// TIA Portal V16 export
FUNCTION_BLOCK "FB_PumpControl_LAD"   // FB2, LAD
{ S7_Optimized_Access := 'TRUE' }
// stored: AutoNumber true
   VAR_INPUT
      FirstScan : Bool;
      AutoMode : Bool;
      StartButton : Bool;
      StopOK : Bool;
      SafetyOK : Bool;
      OverloadOK : Bool;
      SourceWaterOK : Bool;
      LowWet : Bool;
      HighWet : Bool;
      ResetButton : Bool;
      MotorFeedback : Bool;
      MinOffTime : Time := T#5s;
      FeedbackTime : Time := T#3s;
      MaxRunTime : Time := T#10m;
   END_VAR
   VAR_OUTPUT
      PumpCmd : Bool;
      Alarm : Bool;
      Enabled : Bool;
      RunningConfirmed : Bool;
      FaultBits : Word;
      State : USInt;
   END_VAR
   VAR
      RunState : Bool := FALSE;
      EnableState : Bool := FALSE;
      FaultMemory : Word := W#16#0000;
      StartPrev : Bool;
      ResetPrev : Bool;
      AutoPrev : Bool;
      AutoDemand : Bool;
      ManualDemand : Bool;
      OffTimer : TON_TIME;
      RunTimer : TON_TIME;
      StartFeedbackTimer : TON_TIME;
      StopFeedbackTimer : TON_TIME;
   END_VAR
   VAR_TEMP
      StartPulse : Bool;
      ResetPulse : Bool;
      ModeChanged : Bool;
      SensorInvalid : Bool;
      ConfigInvalid : Bool;
      HealthyInputs : Bool;
      Demand : Bool;
      BadMinOff : Bool;
      BadFeedback : Bool;
      BadMaxRun : Bool;
      Disarm : Bool;
      StartAccepted : Bool;
   END_VAR
BEGIN

REGION Network 1: 01 - Startup: reset RunState
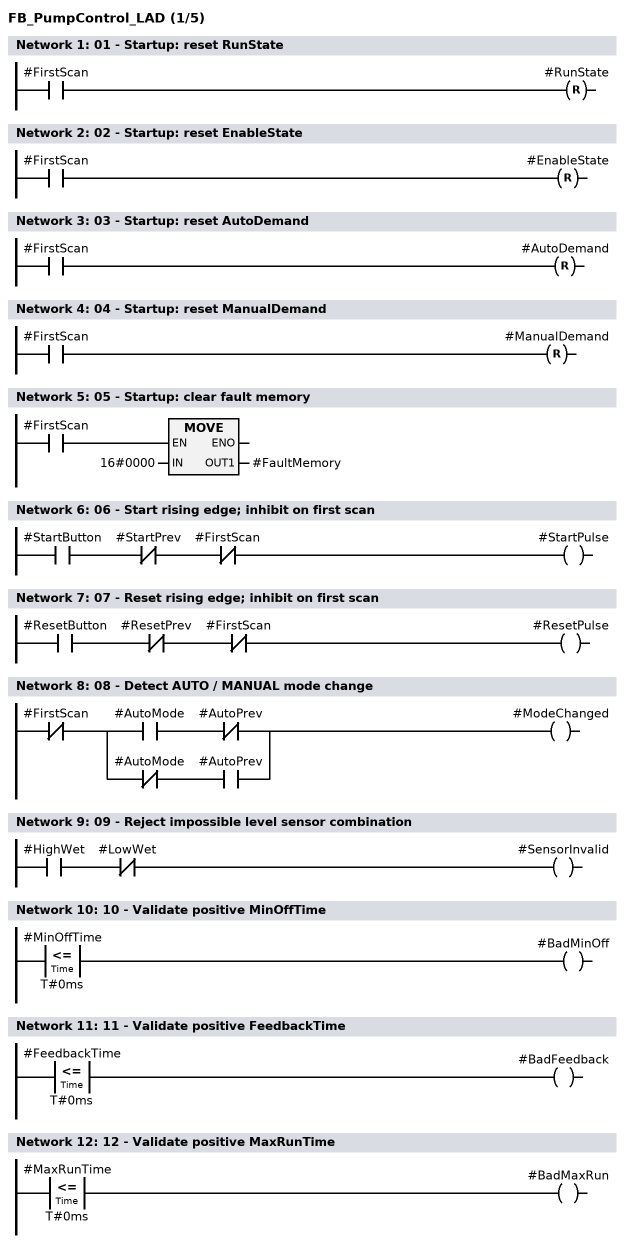
   RUNG wire#powerrail
      Contact( #FirstScan )
      R_Coil( #RunState )
   END_RUNG
   // the same network as SCL:
   IF #FirstScan THEN #RunState := FALSE; END_IF;
END_REGION

REGION Network 2: 02 - Startup: reset EnableState
   RUNG wire#powerrail
      Contact( #FirstScan )
      R_Coil( #EnableState )
   END_RUNG
   // the same network as SCL:
   IF #FirstScan THEN #EnableState := FALSE; END_IF;
END_REGION

REGION Network 3: 03 - Startup: reset AutoDemand
   RUNG wire#powerrail
      Contact( #FirstScan )
      R_Coil( #AutoDemand )
   END_RUNG
   // the same network as SCL:
   IF #FirstScan THEN #AutoDemand := FALSE; END_IF;
END_REGION

REGION Network 4: 04 - Startup: reset ManualDemand
   RUNG wire#powerrail
      Contact( #FirstScan )
      R_Coil( #ManualDemand )
   END_RUNG
   // the same network as SCL:
   IF #FirstScan THEN #ManualDemand := FALSE; END_IF;
END_REGION

REGION Network 5: 05 - Startup: clear fault memory
   RUNG wire#powerrail
      Contact( #FirstScan )
      { S7_GenerateENO := "TRUE" } Move(in := 16#0000, out1 => #FaultMemory)
   END_RUNG
   // the same network as SCL:
   IF #FirstScan THEN #FaultMemory := 16#0000; END_IF;
END_REGION

REGION Network 6: 06 - Start rising edge; inhibit on first scan
   RUNG wire#powerrail
      Contact( #StartButton )
      I_Contact( #StartPrev )
      I_Contact( #FirstScan )
      Coil( #StartPulse )
   END_RUNG
   // the same network as SCL:
   #StartPulse := #StartButton AND NOT #StartPrev AND NOT #FirstScan;
END_REGION

REGION Network 7: 07 - Reset rising edge; inhibit on first scan
   RUNG wire#powerrail
      Contact( #ResetButton )
      I_Contact( #ResetPrev )
      I_Contact( #FirstScan )
      Coil( #ResetPulse )
   END_RUNG
   // the same network as SCL:
   #ResetPulse := #ResetButton AND NOT #ResetPrev AND NOT #FirstScan;
END_REGION

REGION Network 8: 08 - Detect AUTO / MANUAL mode change
   RUNG wire#powerrail
      I_Contact( #FirstScan )
      wire#w1
      Contact( #AutoMode )
      I_Contact( #AutoPrev )
      wire#w2
      Coil( #ModeChanged )
   END_RUNG
   RUNG wire#w1
      I_Contact( #AutoMode )
      Contact( #AutoPrev )
   END_RUNG wire#w2
   // the same network as SCL:
   #ModeChanged := NOT #FirstScan AND ((#AutoMode AND NOT #AutoPrev) OR (NOT #AutoMode AND #AutoPrev));
END_REGION

REGION Network 9: 09 - Reject impossible level sensor combination
   RUNG wire#powerrail
      Contact( #HighWet )
      I_Contact( #LowWet )
      Coil( #SensorInvalid )
   END_RUNG
   // the same network as SCL:
   #SensorInvalid := #HighWet AND NOT #LowWet;
END_REGION

REGION Network 10: 10 - Validate positive MinOffTime
   RUNG wire#powerrail
      { S7_Templates := "SrcType := Time" } LE_Contact(in1 := #MinOffTime, in2 := T#0ms)
      Coil( #BadMinOff )
   END_RUNG
   // the same network as SCL:
   #BadMinOff := #MinOffTime <= T#0ms;
END_REGION

REGION Network 11: 11 - Validate positive FeedbackTime
   RUNG wire#powerrail
      { S7_Templates := "SrcType := Time" } LE_Contact(in1 := #FeedbackTime, in2 := T#0ms)
      Coil( #BadFeedback )
   END_RUNG
   // the same network as SCL:
   #BadFeedback := #FeedbackTime <= T#0ms;
END_REGION

REGION Network 12: 12 - Validate positive MaxRunTime
   RUNG wire#powerrail
      { S7_Templates := "SrcType := Time" } LE_Contact(in1 := #MaxRunTime, in2 := T#0ms)
      Coil( #BadMaxRun )
   END_RUNG
   // the same network as SCL:
   #BadMaxRun := #MaxRunTime <= T#0ms;
END_REGION

REGION Network 13: 13 - Any invalid timer preset
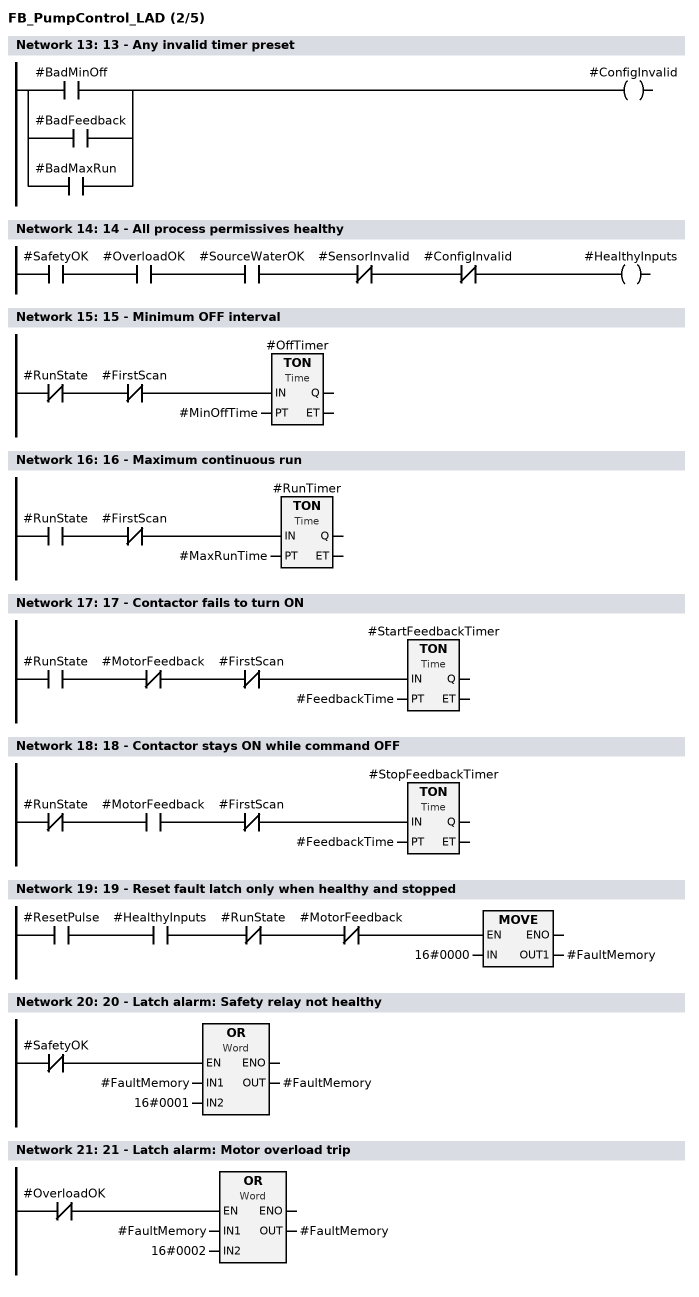
   RUNG wire#powerrail
      Contact( #BadMinOff )
      wire#w1
      Coil( #ConfigInvalid )
   END_RUNG
   RUNG wire#powerrail
      Contact( #BadFeedback )
   END_RUNG wire#w1
   RUNG wire#powerrail
      Contact( #BadMaxRun )
   END_RUNG wire#w1
   // the same network as SCL:
   #ConfigInvalid := #BadMinOff OR #BadFeedback OR #BadMaxRun;
END_REGION

REGION Network 14: 14 - All process permissives healthy
   RUNG wire#powerrail
      Contact( #SafetyOK )
      Contact( #OverloadOK )
      Contact( #SourceWaterOK )
      I_Contact( #SensorInvalid )
      I_Contact( #ConfigInvalid )
      Coil( #HealthyInputs )
   END_RUNG
   // the same network as SCL:
   #HealthyInputs := #SafetyOK AND #OverloadOK AND #SourceWaterOK AND NOT #SensorInvalid AND NOT #ConfigInvalid;
END_REGION

REGION Network 15: 15 - Minimum OFF interval
   RUNG wire#powerrail
      I_Contact( #RunState )
      I_Contact( #FirstScan )
      { S7_Templates := "time_type := Time" } #OffTimer.TON(pt := #MinOffTime, et =>)
   END_RUNG
   // the same network as SCL:
   #OffTimer(IN := NOT #RunState AND NOT #FirstScan, PT := #MinOffTime);   // TON
END_REGION

REGION Network 16: 16 - Maximum continuous run
   RUNG wire#powerrail
      Contact( #RunState )
      I_Contact( #FirstScan )
      { S7_Templates := "time_type := Time" } #RunTimer.TON(pt := #MaxRunTime, et =>)
   END_RUNG
   // the same network as SCL:
   #RunTimer(IN := #RunState AND NOT #FirstScan, PT := #MaxRunTime);   // TON
END_REGION

REGION Network 17: 17 - Contactor fails to turn ON
   RUNG wire#powerrail
      Contact( #RunState )
      I_Contact( #MotorFeedback )
      I_Contact( #FirstScan )
      { S7_Templates := "time_type := Time" } #StartFeedbackTimer.TON(pt := #FeedbackTime, et =>)
   END_RUNG
   // the same network as SCL:
   #StartFeedbackTimer(IN := #RunState AND NOT #MotorFeedback AND NOT #FirstScan, PT := #FeedbackTime);   // TON
END_REGION

REGION Network 18: 18 - Contactor stays ON while command OFF
   RUNG wire#powerrail
      I_Contact( #RunState )
      Contact( #MotorFeedback )
      I_Contact( #FirstScan )
      { S7_Templates := "time_type := Time" } #StopFeedbackTimer.TON(pt := #FeedbackTime, et =>)
   END_RUNG
   // the same network as SCL:
   #StopFeedbackTimer(IN := NOT #RunState AND #MotorFeedback AND NOT #FirstScan, PT := #FeedbackTime);   // TON
END_REGION

REGION Network 19: 19 - Reset fault latch only when healthy and stopped
   RUNG wire#powerrail
      Contact( #ResetPulse )
      Contact( #HealthyInputs )
      I_Contact( #RunState )
      I_Contact( #MotorFeedback )
      { S7_GenerateENO := "TRUE" } Move(in := 16#0000, out1 => #FaultMemory)
   END_RUNG
   // the same network as SCL:
   IF #ResetPulse AND #HealthyInputs AND NOT #RunState AND NOT #MotorFeedback THEN
       #FaultMemory := 16#0000;
   END_IF;
END_REGION

REGION Network 20: 20 - Latch alarm: Safety relay not healthy
   IF NOT #SafetyOK THEN #FaultMemory := #FaultMemory OR 16#0001; END_IF;
END_REGION

REGION Network 21: 21 - Latch alarm: Motor overload trip
   IF NOT #OverloadOK THEN #FaultMemory := #FaultMemory OR 16#0002; END_IF;
END_REGION

REGION Network 22: 22 - Latch alarm: Source water insufficient
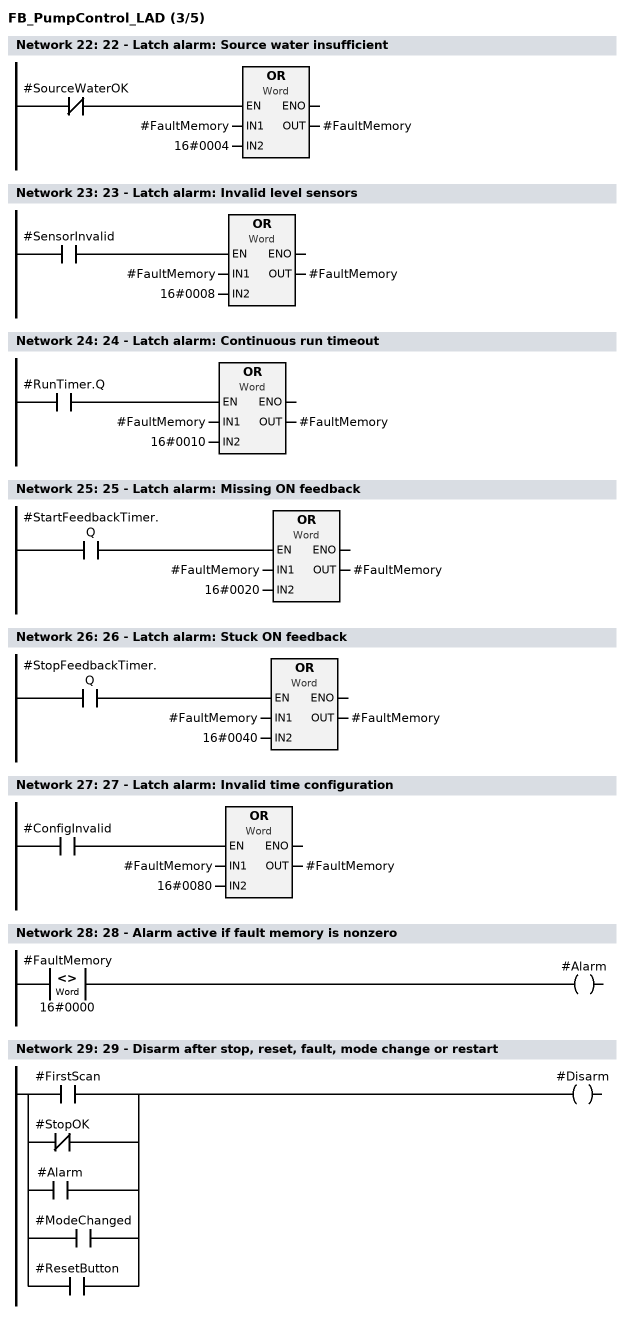
   IF NOT #SourceWaterOK THEN #FaultMemory := #FaultMemory OR 16#0004; END_IF;
END_REGION

REGION Network 23: 23 - Latch alarm: Invalid level sensors
   IF #SensorInvalid THEN #FaultMemory := #FaultMemory OR 16#0008; END_IF;
END_REGION

REGION Network 24: 24 - Latch alarm: Continuous run timeout
   IF #RunTimer.Q THEN #FaultMemory := #FaultMemory OR 16#0010; END_IF;
END_REGION

REGION Network 25: 25 - Latch alarm: Missing ON feedback
   IF #StartFeedbackTimer.Q THEN #FaultMemory := #FaultMemory OR 16#0020; END_IF;
END_REGION

REGION Network 26: 26 - Latch alarm: Stuck ON feedback
   IF #StopFeedbackTimer.Q THEN #FaultMemory := #FaultMemory OR 16#0040; END_IF;
END_REGION

REGION Network 27: 27 - Latch alarm: Invalid time configuration
   IF #ConfigInvalid THEN #FaultMemory := #FaultMemory OR 16#0080; END_IF;
END_REGION

REGION Network 28: 28 - Alarm active if fault memory is nonzero
   RUNG wire#powerrail
      { S7_Templates := "SrcType := Word" } NE_Contact(in1 := #FaultMemory, in2 := 16#0000)
      Coil( #Alarm )
   END_RUNG
   // the same network as SCL:
   #Alarm := #FaultMemory <> 16#0000;
END_REGION

REGION Network 29: 29 - Disarm after stop, reset, fault, mode change or restart
   RUNG wire#powerrail
      Contact( #FirstScan )
      wire#w1
      Coil( #Disarm )
   END_RUNG
   RUNG wire#powerrail
      I_Contact( #StopOK )
   END_RUNG wire#w1
   RUNG wire#powerrail
      Contact( #Alarm )
   END_RUNG wire#w1
   RUNG wire#powerrail
      Contact( #ModeChanged )
   END_RUNG wire#w1
   RUNG wire#powerrail
      Contact( #ResetButton )
   END_RUNG wire#w1
   // the same network as SCL:
   #Disarm := #FirstScan OR NOT #StopOK OR #Alarm OR #ModeChanged OR #ResetButton;
END_REGION

REGION Network 30: 30 - Accept a new Start edge only while healthy
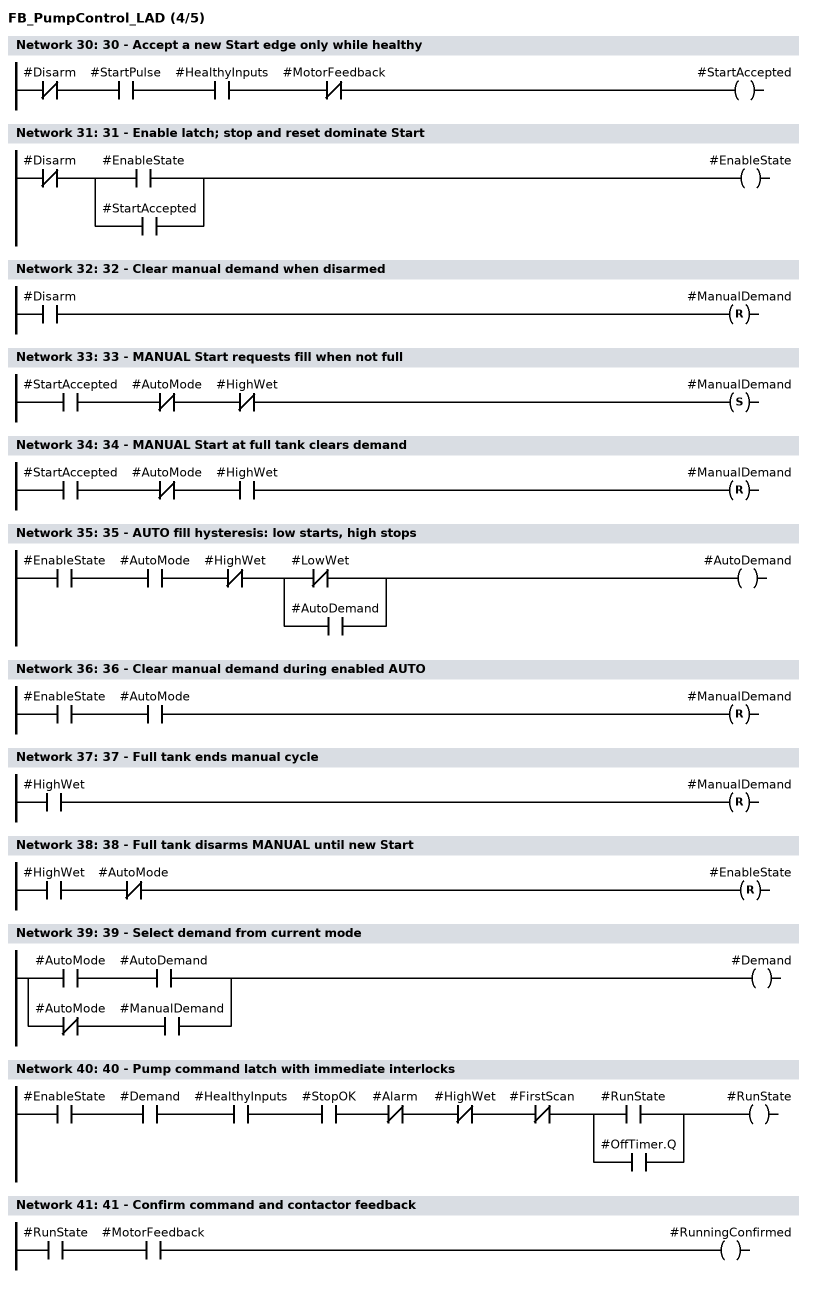
   RUNG wire#powerrail
      I_Contact( #Disarm )
      Contact( #StartPulse )
      Contact( #HealthyInputs )
      I_Contact( #MotorFeedback )
      Coil( #StartAccepted )
   END_RUNG
   // the same network as SCL:
   #StartAccepted := NOT #Disarm AND #StartPulse AND #HealthyInputs AND NOT #MotorFeedback;
END_REGION

REGION Network 31: 31 - Enable latch; stop and reset dominate Start
   RUNG wire#powerrail
      I_Contact( #Disarm )
      wire#w1
      Contact( #EnableState )
      wire#w2
      Coil( #EnableState )
   END_RUNG
   RUNG wire#w1
      Contact( #StartAccepted )
   END_RUNG wire#w2
   // the same network as SCL:
   #EnableState := NOT #Disarm AND (#EnableState OR #StartAccepted);
END_REGION

REGION Network 32: 32 - Clear manual demand when disarmed
   RUNG wire#powerrail
      Contact( #Disarm )
      R_Coil( #ManualDemand )
   END_RUNG
   // the same network as SCL:
   IF #Disarm THEN #ManualDemand := FALSE; END_IF;
END_REGION

REGION Network 33: 33 - MANUAL Start requests fill when not full
   RUNG wire#powerrail
      Contact( #StartAccepted )
      I_Contact( #AutoMode )
      I_Contact( #HighWet )
      S_Coil( #ManualDemand )
   END_RUNG
   // the same network as SCL:
   IF #StartAccepted AND NOT #AutoMode AND NOT #HighWet THEN #ManualDemand := TRUE; END_IF;
END_REGION

REGION Network 34: 34 - MANUAL Start at full tank clears demand
   RUNG wire#powerrail
      Contact( #StartAccepted )
      I_Contact( #AutoMode )
      Contact( #HighWet )
      R_Coil( #ManualDemand )
   END_RUNG
   // the same network as SCL:
   IF #StartAccepted AND NOT #AutoMode AND #HighWet THEN #ManualDemand := FALSE; END_IF;
END_REGION

REGION Network 35: 35 - AUTO fill hysteresis: low starts, high stops
   RUNG wire#powerrail
      Contact( #EnableState )
      Contact( #AutoMode )
      I_Contact( #HighWet )
      wire#w1
      I_Contact( #LowWet )
      wire#w2
      Coil( #AutoDemand )
   END_RUNG
   RUNG wire#w1
      Contact( #AutoDemand )
   END_RUNG wire#w2
   // the same network as SCL:
   #AutoDemand := #EnableState AND #AutoMode AND NOT #HighWet AND (NOT #LowWet OR #AutoDemand);
END_REGION

REGION Network 36: 36 - Clear manual demand during enabled AUTO
   RUNG wire#powerrail
      Contact( #EnableState )
      Contact( #AutoMode )
      R_Coil( #ManualDemand )
   END_RUNG
   // the same network as SCL:
   IF #EnableState AND #AutoMode THEN #ManualDemand := FALSE; END_IF;
END_REGION

REGION Network 37: 37 - Full tank ends manual cycle
   RUNG wire#powerrail
      Contact( #HighWet )
      R_Coil( #ManualDemand )
   END_RUNG
   // the same network as SCL:
   IF #HighWet THEN #ManualDemand := FALSE; END_IF;
END_REGION

REGION Network 38: 38 - Full tank disarms MANUAL until new Start
   RUNG wire#powerrail
      Contact( #HighWet )
      I_Contact( #AutoMode )
      R_Coil( #EnableState )
   END_RUNG
   // the same network as SCL:
   IF #HighWet AND NOT #AutoMode THEN #EnableState := FALSE; END_IF;
END_REGION

REGION Network 39: 39 - Select demand from current mode
   RUNG wire#powerrail
      Contact( #AutoMode )
      Contact( #AutoDemand )
      wire#w1
      Coil( #Demand )
   END_RUNG
   RUNG wire#powerrail
      I_Contact( #AutoMode )
      Contact( #ManualDemand )
   END_RUNG wire#w1
   // the same network as SCL:
   #Demand := (#AutoMode AND #AutoDemand) OR (NOT #AutoMode AND #ManualDemand);
END_REGION

REGION Network 40: 40 - Pump command latch with immediate interlocks
   RUNG wire#powerrail
      Contact( #EnableState )
      Contact( #Demand )
      Contact( #HealthyInputs )
      Contact( #StopOK )
      I_Contact( #Alarm )
      I_Contact( #HighWet )
      I_Contact( #FirstScan )
      wire#w1
      Contact( #RunState )
      wire#w2
      Coil( #RunState )
   END_RUNG
   RUNG wire#w1
      Contact( #OffTimer.Q )
   END_RUNG wire#w2
   // the same network as SCL:
   #RunState := #EnableState AND #Demand AND #HealthyInputs AND #StopOK AND NOT #Alarm AND NOT #HighWet AND NOT #FirstScan AND (#RunState OR #OffTimer.Q);
END_REGION

REGION Network 41: 41 - Confirm command and contactor feedback
   RUNG wire#powerrail
      Contact( #RunState )
      Contact( #MotorFeedback )
      Coil( #RunningConfirmed )
   END_RUNG
   // the same network as SCL:
   #RunningConfirmed := #RunState AND #MotorFeedback;
END_REGION

REGION Network 42: 42 - State default: AUTO standby
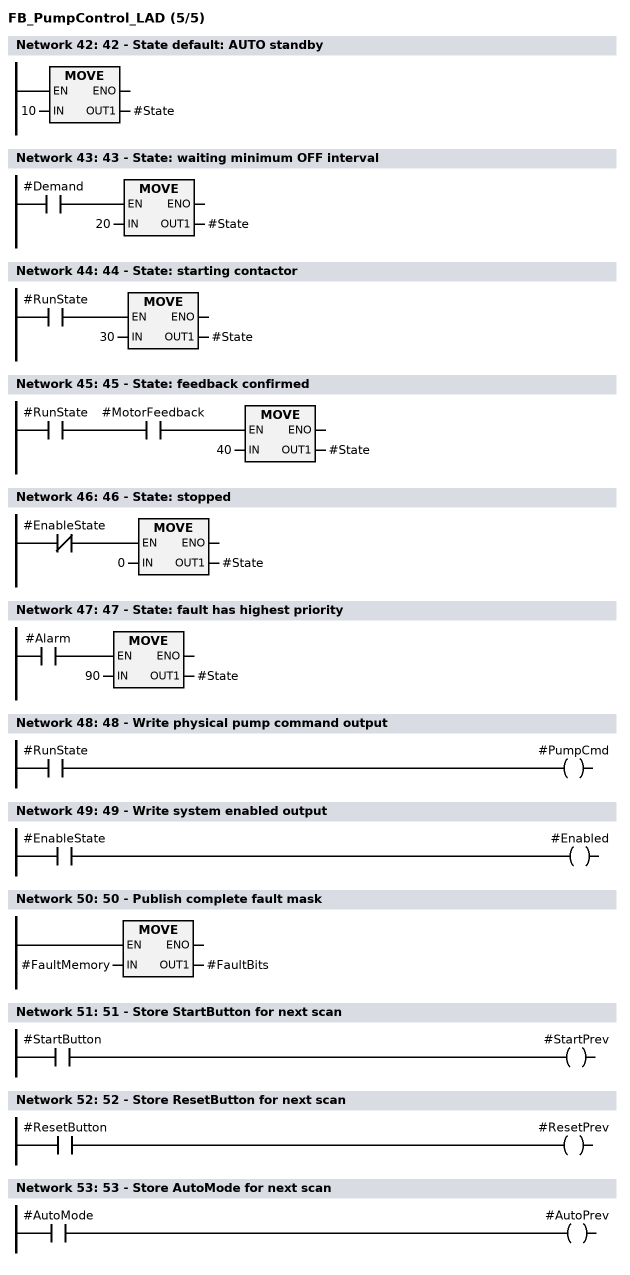
   RUNG wire#powerrail
      { S7_GenerateENO := "TRUE" } Move(in := 10, out1 => #State)
   END_RUNG
   // the same network as SCL:
   #State := 10;
END_REGION

REGION Network 43: 43 - State: waiting minimum OFF interval
   RUNG wire#powerrail
      Contact( #Demand )
      { S7_GenerateENO := "TRUE" } Move(in := 20, out1 => #State)
   END_RUNG
   // the same network as SCL:
   IF #Demand THEN #State := 20; END_IF;
END_REGION

REGION Network 44: 44 - State: starting contactor
   RUNG wire#powerrail
      Contact( #RunState )
      { S7_GenerateENO := "TRUE" } Move(in := 30, out1 => #State)
   END_RUNG
   // the same network as SCL:
   IF #RunState THEN #State := 30; END_IF;
END_REGION

REGION Network 45: 45 - State: feedback confirmed
   RUNG wire#powerrail
      Contact( #RunState )
      Contact( #MotorFeedback )
      { S7_GenerateENO := "TRUE" } Move(in := 40, out1 => #State)
   END_RUNG
   // the same network as SCL:
   IF #RunState AND #MotorFeedback THEN #State := 40; END_IF;
END_REGION

REGION Network 46: 46 - State: stopped
   RUNG wire#powerrail
      I_Contact( #EnableState )
      { S7_GenerateENO := "TRUE" } Move(in := 0, out1 => #State)
   END_RUNG
   // the same network as SCL:
   IF NOT #EnableState THEN #State := 0; END_IF;
END_REGION

REGION Network 47: 47 - State: fault has highest priority
   RUNG wire#powerrail
      Contact( #Alarm )
      { S7_GenerateENO := "TRUE" } Move(in := 90, out1 => #State)
   END_RUNG
   // the same network as SCL:
   IF #Alarm THEN #State := 90; END_IF;
END_REGION

REGION Network 48: 48 - Write physical pump command output
   RUNG wire#powerrail
      Contact( #RunState )
      Coil( #PumpCmd )
   END_RUNG
   // the same network as SCL:
   #PumpCmd := #RunState;
END_REGION

REGION Network 49: 49 - Write system enabled output
   RUNG wire#powerrail
      Contact( #EnableState )
      Coil( #Enabled )
   END_RUNG
   // the same network as SCL:
   #Enabled := #EnableState;
END_REGION

REGION Network 50: 50 - Publish complete fault mask
   RUNG wire#powerrail
      { S7_GenerateENO := "TRUE" } Move(in := #FaultMemory, out1 => #FaultBits)
   END_RUNG
   // the same network as SCL:
   #FaultBits := #FaultMemory;
END_REGION

REGION Network 51: 51 - Store StartButton for next scan
   RUNG wire#powerrail
      Contact( #StartButton )
      Coil( #StartPrev )
   END_RUNG
   // the same network as SCL:
   #StartPrev := #StartButton;
END_REGION

REGION Network 52: 52 - Store ResetButton for next scan
   RUNG wire#powerrail
      Contact( #ResetButton )
      Coil( #ResetPrev )
   END_RUNG
   // the same network as SCL:
   #ResetPrev := #ResetButton;
END_REGION

REGION Network 53: 53 - Store AutoMode for next scan
   RUNG wire#powerrail
      Contact( #AutoMode )
      Coil( #AutoPrev )
   END_RUNG
   // the same network as SCL:
   #AutoPrev := #AutoMode;
END_REGION
END_FUNCTION_BLOCK
